FUNCTION_BLOCK F_MAX (* maximum *)
  (* Standard: 61131-3; Classification: standard selection function; Description: Copyright (c) 2012 TU Wien ACIN This program and the accompanying materials are made available under the terms of the Eclipse Public License 2.0 which is available at https://www.eclipse.org/legal/epl-2.0/ SPDX-License-Identifier: EPL-2.0 *)
  (* Version 1.0, 2012-03-25, Monika Wenger, TU Wien ACIN *)
  (* Version 3.0, 2025-04-14, Patrick Aigner, changed package *)
  PACKAGE iec61131::selection;
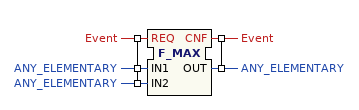
  EVENT_INPUT
    REQ WITH IN1, IN2; (* Service Request *)
  END_EVENT
  EVENT_OUTPUT
    CNF WITH OUT; (* Confirmation of Requested Service *)
  END_EVENT
  VAR_INPUT
    IN1 : ANY_ELEMENTARY; (* Input value 1 *)
    IN2 : ANY_ELEMENTARY; (* Input value 2 *)
  END_VAR
  VAR_OUTPUT
    OUT : ANY_ELEMENTARY; (* maximum value *)
  END_VAR
END_FUNCTION_BLOCK
